TYPE E_Operation :
(
	Addition := 0,
	Substract,
	Multiply,
	Divide
);
END_TYPE

(* stored: Version 1.1.0.1, ProductVersion 3.1.4024.0
   DUT E_Operation: Id {10bcde5b-50bb-474e-9e9d-abaaa27213db} *)
